FUNCTION F_SetProcess : INT
VAR_INPUT
	Process																: INT;
	Mode																: STRING;
END_VAR
VAR
END_VAR

// F_SetProcess
// Rev 1.0 - May 3, 2024

F_SetProcess															:= FIND(INT_TO_STRING(Process), Mode);

END_FUNCTION

(* stored: Version 1.1.0.1, ProductVersion 3.1.4024.12
   POU F_SetProcess: Id {20896656-0d86-4bc2-be72-9eb2d76c3962}, SpecialFunc None *)
